PROGRAM REF_P02_KL1501
VAR
	//bError: BOOL;
	t_1S: TON;	
	
	iStatus: USINT;
	in1: UINT;
	in2: UINT;
		
	encCount: UDINT;
	inData: ST_KL1501InData;
	outData: ST_KL1501OutData;
	KL1501Cfg: FB_KL1501Config;
	
	One_Turn_PLS: REAL ;
	PLS_Old: REAL := 0;
	PLS_New: REAL := 0;
	PLS_Diff: REAL := 0;
	Encoder_Max: REAL := 4294967295; //UINT Range 0 ~ 65,535
	RPM_PV: REAL := 0;
	FB_RPM_AVG: FB_AVG10;
	RPM_AVG: REAL;
    BLDC_MAX_RPM_PLS: REAL := 36000;//genicom : 12PULSE * 3000RPM = 36,000PULSE, china hvpe :500PULSE * 4000RPM = 2,000,000PULSE	
END_VAR

t_1S(PT := T#1S);
t_1S.IN := ON;

//KL1501 Not Use
(*

inData.iState := XA_ENC_ST;
inData.arrDataIn[0] := XA_ENC_IN[0];
inData.arrDataIn[1] := XA_ENC_IN[1];

IF t_1S.Q THEN
	t_1S.IN := Off;
	
	ACT_KL1501();
	
	//Rotation - BLDC Encoder
	pv_ENC := PLS_New := UDINT_TO_REAL(encCount);
	IF N_MAX[29] > 0 THEN
		One_Turn_PLS := BLDC_MAX_RPM_PLS / N_MAX[29];
	ELSE
		One_Turn_PLS := 1;
	END_IF
	IF PLS_New <> PLS_Old THEN //pulse input check
		IF PLS_New <= PLS_Old THEN//Ring counter Check
			PLS_New := PLS_New + Encoder_Max;
		END_IF
		PLS_Diff := PLS_New - PLS_Old;//PLS_Diff is always + value	
		IF PLS_Diff >= 0 THEN	//PLS_Diff is sometime abnormal value
			pv_ROT_inchPulse := pv_ROT_inchPulse + PLS_Diff; //PLS_Diff is always + value
			pv_ROT_1turnPulse := pv_ROT_1turnPulse + PLS_Diff; //PLS_Diff is always + value
			RPM_PV := PLS_Diff * 60 / One_Turn_PLS ;// 60 = 60Sec
		END_IF
		pv_ROT := RPM_PV;
	ELSE	
		pv_ROT := 0;	
	END_IF
	
	IF pv_ROT_1turnPulse >= One_Turn_PLS THEN
		pv_ROT_1turnPulse := pv_ROT_1turnPulse - One_Turn_PLS;
	END_IF
	pv_ROT_DEGREE := pv_ROT_1turnPulse *  360 / One_Turn_PLS;
	
	is_ROT_plsActived := PLS_New <> PLS_Old;
	PLS_Old := PLS_New;	

END_IF;//end 1Sec Timer.Q

*)

ACTION ACT_KL1501:
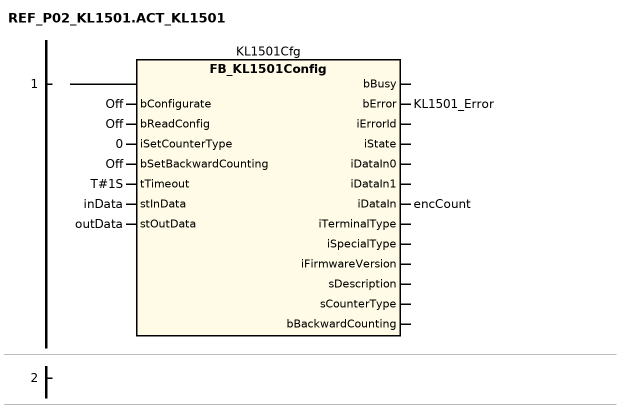
// NETWORK 1
KL1501Cfg(
    bConfigurate := Off,
    bReadConfig := Off,
    iSetCounterType := 0,
    bSetBackwardCounting := Off,
    tTimeout := T#1S,
    stInData := inData,
    stOutData := outData,
    bError => KL1501_Error,
    iDataIn => encCount); // FB_KL1501Config

// NETWORK 2
END_ACTION

END_PROGRAM

(* stored: Version 1.1.0.1, ProductVersion 3.1.4024.12
   POU REF_P02_KL1501: Id {4cfba02f-49ac-45fc-b4b6-ff960cdf1f55}, SpecialFunc None
   Action ACT_KL1501: Id {1199d166-a36a-4b8a-8a1c-b5b527a6c292} *)
